FUNCTION_BLOCK F_COS (* cosine in radians *)
  (* Standard: 61131-3; Classification: standard function of one numeric variable *)
  (* Version 0.0, 2013-04-25, 4DIAC-IDE, 4DIAC-Consortium *)
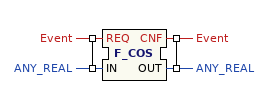
  EVENT_INPUT
    REQ WITH IN; (* Service Request *)
  END_EVENT
  EVENT_OUTPUT
    CNF WITH OUT; (* Confirmation of Requested Service *)
  END_EVENT
  VAR_INPUT
    IN : ANY_REAL; (* Event Input Qualifier *)
  END_VAR
  VAR_OUTPUT
    OUT : ANY_REAL; (* Event Output Qualifier *)
  END_VAR
END_FUNCTION_BLOCK
